// TwinCAT 3 PLC project IBF_Device
// Title: IBF_Device
// Company: Industrial Brains B.V.
// ProjectVersion: 0.0.0.0
// ProgramVersion: 3.1.4022.4
// CompilerDefines: InclSerialCom := 'true'
// libraries:
//   IBF_Utilities, * (Industrial Brains B.V.)
//   Tc2_Math, * (Beckhoff Automation GmbH)
//   Tc2_MC2, * (Beckhoff Automation GmbH)
//   Tc2_MC2_Drive, * (Beckhoff Automation GmbH)
//   Tc2_Standard, * (Beckhoff Automation GmbH)
// project tree:
//   Actuators/Cylinder/DataTypes/ E_CylinderCmd.TcTLEO, E_ValveResetState.TcTLEO (not stored)
//   Actuators/Cylinder/DataTypes/ManualControls/ UDT_ManualValveControl.TcDUT
//   Actuators/Cylinder/Functions/ Fb_DevCylWithFbk.TcPOU (not stored), FB_DevValve.TcPOU (not stored)
//   Axis/DataTypes/ E_AxisCmd.TcTLEO, UDT_AxisData.TcDUT, UDT_AxVal.TcDUT (not stored), UDT_ManualAxisCtrl.TcDUT (not stored)
//   Axis/FunctionBlocks/Analog/ FB_DevAnalogAxis.TcPOU (not stored), ST_ManualAnalogAxisCtrl.TcDUT (not stored)
//   Axis/FunctionBlocks/ServoHybrid/ FB_DevBasicACAxis.TcPOU (not stored), FB_DevHybridAc.TcPOU
//   Axis/FunctionBlocks/Servo/ Fb_DevAxis.TcPOU (not stored)
//   Axis/FunctionBlocks/TwoVelocityControl/DataTypes/ st_ManualDigitalMotorControl.TcDUT (not stored)
//   Axis/FunctionBlocks/TwoVelocityControl/ FB_DevTwoVelocityAxis.TcPOU (not stored)
//   Axis/Interface/ iTwoDirectionalMotor.TcIO (not stored), iTwoDirectionalMotorWithFast.TcIO
//   BaseFunctions/ FB_DevBase.TcPOU (not stored), UDT_DevManualCtrl.TcDUT (not stored)
//   Buttons/Functions/ FB_DevHMIButton.TcPOU, FB_DevPushbuttonLight.TcPOU, FB_DevPushButton.TcPOU
//   CounterCards/FunctionBlocks/KL1512/ FB_DevKL1512.TcPOU (not stored)
//   CounterCards/FunctionBlocks/KL5151/ FB_DevKL5151.TcPOU (not stored)
//   CounterCards/Interfaces/ iCounter.TcIO
//   CounterCards/ st_ManualCounterControl.TcDUT (not stored)
//   DevTypes/ E_Devices.TcTLEO (not stored)
//   Encoders/FunctionBlocks/ FB_EncoderBase.TcPOU (not stored), FB_EncoderInput.TcPOU (not stored)
//   GroupHandlers/ GVL_DevManual.TcGVL (not stored)
//   GroupHandlers/ManualControlHandler/ FB_ManualController.TcPOU (not stored), UDT_DeviceID.TcDUT (not stored)
//   HardwareDiagnostics/ FB_ELModuleDiag.TcPOU (not stored)
//   Heaters/ FB_DevDoublePWM.TcPOU (not stored), FB_DevPWMGenerator.TcPOU (not stored)
//   Lights/Functions/ Fb_DevLight.TcPOU
//   Outputs/AnalogOutputs/ FB_DevAnalogOutput.TcPOU, FB_DevAnalogOutputScaled.TcPOU (not stored)
//   Outputs/DigitalOutputs/ FB_DevDigitalOutput.TcPOU (not stored)
//   Sensors/AnalogInput/FunctionBlocks/ FB_DevAnalogInput.TcPOU (not stored), FB_DevAnalogInputScaled.TcPOU (not stored), FB_DevHDAnalogInAutoCalibrate.TcPOU (not stored), FB_DevAnalogInAutoCalibrate.TcPOU (not stored), FB_DevHDAnalogInputScaled.TcPOU, FB_DevHDAnalogInput.TcPOU (not stored)
//   Sensors/DigitalSensor/FunctionBlocks/ Fb_DevDigitalInput.TcPOU, Fb_DevDigitalInputFunctions.TcPOU (not stored)
//   Sensors/FootPedals/DataTypes/ E_FootpedalPos.TcTLEO (not stored)
//   Sensors/FootPedals/FunctionBlocks/ FB_EfkaEB301A_FootPedal.TcPOU (not stored)
//   Sensors/ModuleSpecific/EL3556_Loadcell/ Fb_DevEL3356_LoadCell.TcPOU
//   Version/ Global_Version.TcGVL

// ---- Actuators/Cylinder/DataTypes/E_CylinderCmd.TcTLEO
(* cylinder commands *)
TYPE E_CylinderCmd :
(
	Cyl_Idle 		:= 0,// Jog Cylinder command Referance 0 Idle (wait for command)
	Cyl_Init 		:= 1,// Jog Cylinder command Referance 1 initialize Cylinder
	Cyl_Enable 		:= 2,// Jog Cylinder command Referance 2 enable
	Cyl_Disable 	:= 3,// Jog Cylinder command Referance 3 disable
	Cyl_Reset 		:= 4,// Jog Cylinder command Referance 4 reset
	Cyl_Hold 		:= 5,// Jog Cylinder command Referance 5 hold
	Cyl_Teach 		:= 6,// Jog Cylinder command Referance 6 teach timeout settings
	Cyl_Calculate 	:= 7,// Jog Cylinder command Referance 7 calculate timeout settings from parameters
	Cyl_Expand 		:= 8,// Jog Cylinder command Referance 8 expand
	Cyl_Retract 	:= 9 // Jog Cylinder command Referance 9 retract
);
END_TYPE

// ---- Actuators/Cylinder/DataTypes/ManualControls/UDT_ManualValveControl.TcDUT
TYPE UDT_ManualValveControl extends UDT_DevManualCtrl:
STRUCT
	// Device commands
	bCmdOpen	: BOOL	; // open valve 
	bCmdClose	: BOOL	; // Close valve
	bCmdTeach	: BOOL	; // Teach valve
END_STRUCT
END_TYPE

// ---- Axis/DataTypes/E_AxisCmd.TcTLEO
(* axis command structure *)
TYPE E_AxisCmd :
(
	Ax_Idle 		:= 0,// Axis command Referance 0 Axis Idle
	Ax_Init 		:= 1,// Axis command Referance 1 Initialize axis
	Ax_Enable 		:= 2,// Axis command Referance 2 Enable
	Ax_Disable 		:= 3,// Axis command Referance 3 Disable
	Ax_Reset 		:= 4,// Axis command Referance 4 Reset
	Ax_Hold 		:= 5,// Axis command Referance 5 Hold
	Ax_Home 		:= 6,// Axis command Referance 6 Home
	Ax_JogFwd 		:= 7,// Axis command Referance 7 Jog Forward
	Ax_JogRev 		:= 8,// Axis command Referance 8 Jog Reverse
	Ax_MoveRelative := 9,// Axis command Referance 9 Move axis relative
	Ax_MoveAbs 		:= 10,// Axis command Referance 11 Move absolute reverse
	Ax_MoveModulo 	:= 11,// Axis command Referance 11 Move Module
	Ax_MoveVeloFwd 	:= 12,// Axis command Referance 12 Move velocity forward
	Ax_MoveVeloRev 	:= 13,// Axis command Referance 13 Move velocity reverse
	Ax_HardStop 	:= 14,// Axis command Referance 14 hard stop or emergency stop
	Ax_SoftStop 	:= 15,// Axis command Referance 15 soft stop after motion command
	Ax_GearSlave 	:= 16,// Axis command Referance 16 gear axis as slave
	Ax_GearSlaveDyn	:= 17,// Axis command Referance 17 gear axis as slave dynamic
	Ax_GearOutSlave := 18,// Axis command Referance 18 gear out from Master axis 
	Ax_Maintenance	:= 50 // Axis Command referance 50 maintenance mode, axis enabled with no command active
);
END_TYPE

// ---- Axis/DataTypes/UDT_AxisData.TcDUT
TYPE UDT_AxisData:
STRUCT
	// ===== Axis name =====
		AxisName	: STRING 	; // Name of the axis (used for fault handling and identification)
		AxisNumber	: INT		; // Axis number 

	// ===== Fault data =====
		Message			: UDT_Fault 	; // Message data from Cylinder
		MessageActive	: BOOL			; // Message is active
		ErrorActive 	: BOOL 			;	// Axis in error state

	// ===== Axis Commands =====
		// ***** Enable command	*****
			CmdEnable		: BOOL 		; // Command enable axis
		// ***** Active commands *****
			AxisCmd			: E_AxisCmd ; // Axis command
			AxisSafeCmd		: E_AxisCmd	; // Axis safe command
			AxisAct			: E_AxisCmd ; // Axis Active status
		// ***** Command Modes *****
			CmdHomingMode 	: MC_HomingMode ; // Homing Mode ( MC_DefaultHoming, MC_Direct, MC_ForceCallibration, MC_ResetCallibration)
			CmdJogMode		: E_JogMode 	;
			CmdBuffermode	: MC_BufferMode	; // Buffermode used for command transition 	 
	// ===== Axis Safe commands =====
		SafeCmdLimitVelo: BOOL 	; // safe command limit velocity
		SafeCmdVelocity	: LREAL ; // Safe command velocity
		SafeCmdStop		: BOOL 	; // Stop command from safety or collision detection		
		SafeVeloLimit	: LREAL ; // safe velocity limit (link to FPAR)
	// ===== Status indication active =====
		ActHoming	: BOOL ; // Axis is homing
		ActBusy		: BOOL ; // Axis is Busy 
		ActMoving	: BOOL ; // Axis is moving
		ActAtVelo	: BOOL ; // Axis is at command velocity (only when written in Move velocity mode)

	// ===== Status indication done  =====
		FcoInit		: BOOL ; // Axis is initialised
		FcoIdle		: BOOL ; // Axis is idle enable required
		FcoEnabled	: BOOL ; // Axis is enabled
		FcoHomed	: BOOL ; // Axis is homed
		FcoGeared	: BOOL ; // Axis is geared to master axis
		FcoHeld		: BOOL ; // Axis is holding
		FcoStopped	: BOOL ; // Axis is stopped
		FcoReset	: BOOL ; // Axis reset done
		FcoReady 	: BOOL ; // Axis is ready for command
		FcoAtCmdPos	: BOOL ; // Axis is at command position (tol 0.2 deg)
		FcoCmdActive: BOOL ; // Axis new command values are active
		
	// ===== Move values =====
		Pos			: UDT_Axval	; // possition values (0 = infinite)
		Velocity 	: UDT_AxVal	; // Velocity values
		Accel		: UDT_Axval ; // Aceleration values
		Decel		: UDT_Axval ; // Deceleration values
		Torque		: UDT_Axval ; // Torque values
		EncTurnoverVal	: DINT 	; // Encoder turnover value
		TimeDisableDelay : TIME ; // Time off delay after axis move command (remove enable)
		
	// ===== Config Bits =====
		IcfCommandSpeedRpm	: BOOL ; // input speeds in Rpm
		IcfEnableForward 	: BOOL ; // Enable forward motion
 		IcfEnablereverse	: BOOL ; // Enable reverse motion
		IcfContinuous		: BOOL ; // continuous motion possible (no endpoint)
		IcfAlwaysEnable		: BOOL ; // 1 = Axis always enabled, 0 = Axis disabled at Idle 
		
	// ===== Master Axis =====
		MasterAxisRef	: REFERENCE TO AXIS_REF ; // Master axis reference (if applicable)
		GearMasterRev	: UINT	:= 1	; // Master Axis Gearing revolutions (Denominator)
		GearSlaveRev	: LREAL	:= 1	; // Slave Axis gearing revolutions (numerator)	
		ReverseSlave	: BOOL 	; // Reverse slave axis relative to master
		 
END_STRUCT
END_TYPE

// ---- Version/Global_Version.TcGVL
{attribute 'TcGenerated'}
{attribute 'no-analysis'}
{attribute 'linkalways'}
// This function has been automatically generated from the project information.
VAR_GLOBAL CONSTANT
	{attribute 'const_non_replaced'}
	stLibVersion_IBF_Device : ST_LibVersion := (iMajor := 0, iMinor := 0, iBuild := 0, iRevision := 0, nFlags := 0, sVersion := '0.0.0.0');
END_VAR

// ---- Axis/Interface/iTwoDirectionalMotorWithFast.TcIO
INTERFACE iTwoDirectionalMotorWithFast EXTENDS iTwoDirectionalMotor // Two directional motor with run fast commands

METHOD CmdRunCCWFast : BOOL
VAR_INPUT
END_VAR
END_METHOD

METHOD CmdRunCWFast : BOOL
VAR_INPUT
END_VAR
END_METHOD

END_INTERFACE

// ---- CounterCards/Interfaces/iCounter.TcIO
INTERFACE iCounter

METHOD PUBLIC CmdResetValue : BOOL
END_METHOD

METHOD PUBLIC CmdSetValue : BOOL
VAR_INPUT
	Value : UDINT ;
END_VAR
END_METHOD

PROPERTY PUBLIC CountValue : UDINT
GET
END_GET
END_PROPERTY

END_INTERFACE

// ---- Axis/FunctionBlocks/ServoHybrid/FB_DevHybridAc.TcPOU
{attribute 'reflection'}
FUNCTION_BLOCK PUBLIC FB_DevHybridAc EXTENDS Fb_DevAxis
VAR_INPUT
END_VAR
VAR_OUTPUT
END_VAR
VAR
	// Parameters 
		stMParMaxAcc : Udt_Parameter := (fMaximum := 999999, fMinimum := 0, fValue := 0)	; // Parameter for maximum acceleration
		stMParMaxDec : Udt_Parameter := (fMaximum := 999999, fMinimum := 0, fValue := 0)	; // Parameter for maximum Deceleration
		stMparMaxVelo: Udt_Parameter := (fMaximum := 999999, fMinimum := 0, fValue := 0)	; // Parameter for maximum velocity
END_VAR

SUPER^(refFbFault := refFbFault);

METHOD INTERNAL ExecHalt : BOOL
VAR_INPUT
END_VAR
// The hybrid axis is equiped with it's own safety stop system therefore mc halt is no longer needed with an Estop
IF bSafetyOk THEN 
	// ==== Execute halt function ===== 
	fbMcHalt (	Axis 		:= AxisRef,
				Execute 	:= bExec_Halt );
END_IF
// ===== reset command =====
	bExec_Halt := FALSE ;
	
// Halt fault handling 
	IF fbMcHalt.Error THEN 
		bError					:= TRUE							;
		stFault.Active 			:= TRUE 						;
		stFault.MessageNumber	:= E_MessageNumbers.FF_AxisFault;
		stFault.Discription		:= CONCAT('Halt Fault ', UDINT_TO_STRING(fbMcHalt.ErrorID));				;
		stFault.FaultType		:= E_FaultTypes.FF				;
	END_IF
END_METHOD

METHOD INTERNAL ExecReadStatus : BOOL
VAR_INPUT
END_VAR
// Read axis status from drive
AxisRef.ReadStatus();						
// convert velocity to RPM for output if aplicable
IF bIcfCmdVelocityRpm THEN 
	fVelocity := AxisRef.NcToPlc.ActVelo / 6 ;
ELSE 
	fVelocity := AxisRef.NcToPlc.ActVelo ;
END_IF

// write position output
fActPosition := AxisRef.NcToPlc.ActPos ;
						
// set status bits 
bIdle := NOT AxisRef.Status.HasJob ;
END_METHOD

METHOD INTERNAL ExecReset : BOOL
VAR_INPUT
END_VAR
IF  AxisRef.Status.Moving AND bExec_Reset THEN // If the axis is still moving execute safe stop first
	CmdSafeStop();
	RETURN;
END_IF

	fbMcReset	( 	Execute	:= bexec_reset,
					Axis	:= AxisRef ); 
					
// ===== reset command =====
	bExec_Reset := FALSE ;
	
// ===== reset internal fault bits and stop bits =====
	bError 			:= FALSE ; 
	
// ===== reset safe commands ======
	bCmdSafeStop	:= FALSE ; 
	bCmdSafeSpeed 	:= FALSE ;
	
// Reset fault handling 
	IF fbMcReset.Error THEN 
		bError					:= TRUE							;
		stFault.Active 			:= TRUE 						;
		stFault.MessageNumber	:= E_MessageNumbers.FF_AxisFault;
		stFault.Discription		:= CONCAT('Reset Fault ', UDINT_TO_STRING(fbMcReset.ErrorID))			;
		stFault.FaultType		:= E_FaultTypes.FF				;
	END_IF
END_METHOD

METHOD PUBLIC Init : BOOL
VAR_INPUT
	// Message location data
	nId			: UDINT ; // Identification number of object
	nParentId	: UDINT ; // Id of higher level If aplicable (0 = no parent)
	// Config Bits
	bIcfCmdVelocityRpm	: BOOL := FALSE ; // input speeds in Rpm
	bIcfEnableForward 	: BOOL := TRUE 	; // Enable forward motion
	bIcfEnablereverse	: BOOL := TRUE 	; // Enable reverse motion
	bIcfAlwaysEnable	: BOOL := FALSE ; // 1 = Axis always enabled, 0 = Axis disabled at Idle 
	bIcfSimulationMode	: BOOL := FALSE ; // Simulation mode is active [default set to False] Used for testing without hardware present 
	bIcfModuloAxis		: BOOL := FALSE ; // Show axis position as modulo
	bIcfSTOPresent		: BOOL := FALSE ; // Axis safe torque off is present	
	bIcfNCHomeSensor	: BOOL := FALSE ; // Homing sensor is inverted (NC)	

	// Config Values 
	mcHomingMode 		: MC_HomingMode := MC_HomingMode.MC_DefaultHoming; 
	fHomePosition		: LREAL := 0 	; // set position at homing
	fSafeOverride		: LREAL := 10	; // Safe velocity override [%]
	nEncTurnoverVal 	: LREAL := 360	; // encoder turnover value 
	tEnableDelay		: time 	:= T#0MS; // Time between axis enable command and motion command execution (0 := no delay active)	
	tDisabledelay		: TIME 	:= T#100MS; // Axis idle time before axis is disabled 
END_VAR
VAR 
	bActVeloReadValid 	: BOOL ; // velocity parameter read is valid 
	bActAccReadValid 	: BOOL ; // Acceleration parameter read is valid 
	bActDecReadValid 	: BOOL ; // Deceleration parameter read is valid 
	bActParamValid 		: BOOL ; // Parameter read is valid 
END_VAR
// Calculate device number
	ExecIdentifyDevice(nId,nParentId, E_ComponentTypes.Axis);

// ===== Message data set =====
	stFault.ComponentType		:= E_ComponentTypes.Axis ;
	
// ===== Write parameters =====
	stMParMaxAcc.nNumber		:= nLocationId + 1;
	stMParMaxAcc.sDiscription 	:= CONCAT(STR1 := sName, STR2:= ' hardware maximum accaleration (0 = HWMaximum)'); 
	stMParMaxAcc.sName			:= CONCAT(STR1 := sName, STR2:= 'Hard max aceleration');
	stMParMaxAcc.sType			:= 'MPar';
	stMParMaxAcc.sUnit			:= 'Units/Sec^2';
	
	stMParMaxDec.nNumber		:= nLocationId + 2;
	stMParMaxDec.sDiscription 	:= CONCAT(STR1 := sName, STR2:= ' hardware maximum deceleration(0 = HWMaximum)'); 
	stMParMaxDec.sName			:= CONCAT(STR1 := sName, STR2:= 'Hard max deceleration');
	stMParMaxDec.sType			:= 'MPar';
	stMParMaxDec.sUnit			:= 'Units/Sec^2';
	
	stMparMaxVelo.nNumber		:= nLocationId + 3;
	stMparMaxVelo.sDiscription 	:= CONCAT(STR1 := sName, STR2:= ' hardware maximum velocity'); 
	stMparMaxVelo.sName			:= CONCAT(STR1 := sName, STR2:= 'Hard max velocity');
	stMparMaxVelo.sType			:= 'MPar';
	stMparMaxVelo.sUnit			:= 'Units/Sec';

	refFbParHandler.CmdAddParameter(refParameter := stMParMaxAcc);
	refFbParHandler.CmdAddParameter(refParameter := stMParMaxDec);
	refFbParHandler.CmdAddParameter(refParameter := stMparMaxVelo);

// ===== set axis configuration =====	
	fMaxAcc	:= stMParMaxAcc.fValue;
	fMaxDec	:= stMParMaxDec.fValue;	
	fMaxVelo:= stMparMaxVelo.fValue;

	fCmdAcc 		:= fMaxAcc;
	fCmdDecc		:= fMaxDec;
// ===== Configure Axis =====
	// ***** Config Bits *****
		THIS^.bIcfCmdVelocityRpm	:= bIcfCmdVelocityRpm	; // Enable speed inputs in Rpm
		THIS^.bIcfEnableForward 	:= bIcfEnableForward 	; // Enable forward motion
		THIS^.bIcfEnablereverse		:= bIcfEnablereverse	; // Enable reverse motion
		THIS^.bIcfAlwaysEnable		:= bIcfAlwaysEnable		; // Always enable motor and brake if safety is ok
		THIS^.bIcfSimulationMode	:= bIcfSimulationMode 	; // Simulation mode is active [default set to False] 

	// ***** config homing Mode ***** 
 		THIS^.mcHomingMode 			:= mcHomingMode ; // set homing mode
 		THIS^.fHomePosition			:= fHomePosition;
	// ***** Velocity settings *****
		THIS^.fSafeOverride			:= fSafeOverride	; 	
	// ***** Time delay enable off *****
		THIS^.tEnableDelay		:= tEnableDelay	;
		THIS^.tDisableDelay 	:= tDisabledelay ;		

// ===== Set device type for manual control =====
	eDevType := E_Devices.Axis ;
		
// ===== reset axis state indicators ======
	bErrorActive 	:= FALSE;

// ====== Set init to done =======
	bInitOk	:= TRUE ;
END_METHOD

END_FUNCTION_BLOCK

// ---- Buttons/Functions/FB_DevHMIButton.TcPOU
{attribute 'reflection'}
FUNCTION_BLOCK PUBLIC FB_DevHMIButton EXTENDS FB_DevBase // Button function for HMI 
VAR_INPUT
	Istatus			: BOOL	:= FALSE;// Digital sensor, Direct input status
	tDelay			: TIME 	:= T#5S	;// Time before delayed signal becomes active 
END_VAR
VAR_OUTPUT
	bFcoInputActive		: BOOL 			;// Digital sensor, Button active state
	bFcoDelay			: BOOL			;// Button, Delayed input status (3 seconds) 
	bFeStatus			: BOOL			;// Button, Falling edge of input signal	
	bReStatus			: BOOL			;// Button, Rising edge of input signal
	TetInputActive		: TIME			;// Button, Time elapsed while button is active
	bInvisible			: BOOL 			;// Button, Button is made invisible
	bDeactivate			: BOOL 			;// Button, Deactivate button 
END_VAR
VAR
	FB_delIStatus	: TON; // Timer function for delayed input status 
	FB_feIStatus	: F_TRIG; // generate falling edge pulse edge from Istatus
	FB_reIStatus	: R_TRIG; // generate falling edge pulse edge from Istatus
END_VAR

// Call base function
SUPER^(refFbFault := refFbFault);

// ***** Direct input when enabled *****
IF bEnable THEN 
	bFcoInputActive := Istatus ;
ELSE 
	bFcoInputActive := FALSE ;
END_IF

// ===== check if function is enabled =====
	IF NOT bEnable THEN 
		bInvisible 	:= TRUE ;
		bDeactivate	:= TRUE ;
		bFcoDelay	:= FALSE;
		RETURN;
	ELSE  
		bInvisible 	:= FALSE ;
		bDeactivate	:= FALSE ;
	END_IF

// ====== process functions if enabled ======
	// ***** Set Delayed inputs and time elapsed ****
		FB_delIStatus(	IN:= bFcoInputActive,
						PT:= tDelay , 
						Q=> bFcoDelay , 
						ET=> TetInputActive 
					  ); // Generate delayed input status from push button input status
	// ***** Edge triggers *****
		FB_feIStatus(CLK:= Istatus , Q=> bFeStatus ); // generate falling edge pulse on pushbutton input
		FB_reIStatus (Clk := Istatus , Q => bReStatus); // Generate rising edge from push button input signal

END_FUNCTION_BLOCK

// ---- Buttons/Functions/FB_DevPushbuttonLight.TcPOU
{attribute 'reflection'}
FUNCTION_BLOCK PUBLIC FB_DevPushbuttonLight EXTENDS Fb_DevDigitalInputFunctions
VAR_OUTPUT
END_VAR
VAR
	fbLight : Fb_DevLight ; // light control 
END_VAR

// Set device type
IF eDevType = E_Devices.Undefined THEN 
	eDevType := E_Devices.PushButtonLight ;
END_IF

SUPER^(refFbFault := refFbFault);

// Light commands
	
fbLight(bEnable := bEnable, refFbFault := refFbFault);

METHOD PUBLIC CmdBlinkFast : BOOL
VAR_INPUT
END_VAR
CmdBlinkFast := fbLight.CmdBlinkFast();
END_METHOD

METHOD PUBLIC CmdBlinkSlow : BOOL
VAR_INPUT
END_VAR
CmdBlinkSlow	:= fbLight.CmdBlinkSlow();
END_METHOD

METHOD PUBLIC CmdOn : BOOL
VAR_INPUT
END_VAR
CmdOn := fbLight.CmdOn() ;
END_METHOD

END_FUNCTION_BLOCK

// ---- Lights/Functions/Fb_DevLight.TcPOU
{attribute 'reflection'}
FUNCTION_BLOCK PUBLIC Fb_DevLight EXTENDS FB_DevBase ;
VAR_OUTPUT
	bSoftLightOut	: BOOL ; // Software light output	
END_VAR
VAR
	bCmdBlinkSlow	: BOOL := FALSE ; // Command light blink slow
	bCmdBlinkFast 	: BOOL := FALSE ; // Command light blink fast
	bCmdOn			: BOOL := FALSE ; // Command turn light on	 
	qLight AT %Q* 	: BOOL := FALSE ; // light output
END_VAR

// set device type
IF eDevType = E_Devices.Undefined THEN 
	eDevType := E_Devices.DigitalOut ;
END_IF

// ===== check if light is enabled ======
	IF NOT bEnable AND NOT bCmdManual THEN 
		qLight := FALSE ;
		RETURN; 
	END_IF
	
// ===== set light output ======
	ExecSetOutput();

METHOD PUBLIC CmdBlinkFast : BOOL
VAR_INPUT
END_VAR
bCmdBlinkFast S= TRUE ;

CmdBlinkFast := bCmdBlinkFast ;
END_METHOD

METHOD PUBLIC CmdBlinkSlow : BOOL
VAR_INPUT
END_VAR
bCmdBlinkSlow S= TRUE ;

CmdBlinkSlow	:= bCmdBlinkSlow ;
END_METHOD

METHOD PUBLIC CmdOn : BOOL
VAR_INPUT
END_VAR
bCmdOn S= TRUE ;

CmdOn := qLight ;
END_METHOD

METHOD PRIVATE ExecSetOutput : BOOL
VAR_INPUT
END_VAR
// ===== set light output state =====
IF bCmdOn THEN 
	qLight S= TRUE ;
ELSIF bCmdBlinkFast THEN 
	qLight := Sys_Variables.BlinkFast 	;
ELSIF bCmdBlinkSlow THEN 
	qLight := Sys_Variables.BlinkSlow	;
ELSE
	qLight := FALSE ;
END_IF

// set soft output
bSoftLightOut	:= qLight;

// reset all commands 
bCmdOn			:= FALSE ;
bCmdBlinkFast 	:= FALSE ;
bCmdBlinkSlow 	:= FALSE ;
END_METHOD

METHOD PUBLIC Init : BOOL
VAR_INPUT
	// Location data for messages  
	nId			: UDINT ; // Identification number of object
	nParentId	: UDINT ; // Id of higher level If aplicable (0 = no parent)
END_VAR
// ====== Set init to true =====
	bInitOk	:= TRUE ; 

// ====== Calculate device id =====
	bInitOk :=	ExecIdentifyDevice(nId,nParentId, E_ComponentTypes.DiOutput) AND bInitOk;

// ===== Set feedback =====
	Init := bInitOk;
END_METHOD

END_FUNCTION_BLOCK

// ---- Buttons/Functions/FB_DevPushButton.TcPOU
{attribute 'reflection'}
FUNCTION_BLOCK PUBLIC FB_DevPushButton EXTENDS Fb_DevDigitalInputFunctions
VAR_INPUT
END_VAR
VAR_OUTPUT
END_VAR
VAR
END_VAR

// set device type
IF eDevType = E_Devices.Undefined THEN 
	eDevType := E_Devices.DigitalSensor ;
END_IF

SUPER^(refFbFault := refFbFault);

END_FUNCTION_BLOCK

// ---- Outputs/AnalogOutputs/FB_DevAnalogOutput.TcPOU
{attribute 'reflection'}
FUNCTION_BLOCK PUBLIC FB_DevAnalogOutput EXTENDS FB_DevBase 
VAR_INPUT
	fCmdValue		: LREAL := 0 ;
END_VAR
VAR_OUTPUT
	fOutputValue	: LREAL := 0 ;
END_VAR
VAR
	nLimitMin		: INT := -32767 ;
	nLimitMax 		: INT := 32767 ;
	qnHwOut	AT%Q*	: INT := 0 ;
END_VAR

// set device type
IF eDevType = E_Devices.Undefined THEN 
	eDevType := E_Devices.AnalogOut ;
END_IF

// Call base function
SUPER^(refFbFault := refFbFault);


// Call private functions
ExecSetOutput();
ExecSetFeedback();

METHOD INTERNAL ExecSetFeedback : BOOL
VAR_INPUT
END_VAR
// Set feedback 
fOutputValue := INT_TO_LREAL(qnHwOut) ;
END_METHOD

METHOD INTERNAL ExecSetOutput : BOOL
VAR_INPUT
END_VAR
// Set Output to physical device
IF bSafetyOk AND (bEnable OR bCmdManual) THEN 
	qnHwOut := LREAL_TO_INT(fCmdValue) ; 
	qnHwOut := LIMIT(nLimitMin, qnHwOut, nLimitMax) ; 
ELSE 
	qnHwOut 	:= 0;
	fCmdValue 	:= 0 ; 
END_IF
END_METHOD

METHOD PUBLIC Init : BOOL
VAR_INPUT
	// Location data for messages  
	nId				: UDINT; // Identification number of object
	nParentId		: UDINT; // Id of higher level If aplicable (0 = no parent)
	benableNegative	: BOOL ; // Enable negative values
END_VAR
// ====== Set init to true =====
	bInitOk	:= TRUE ; 

// ====== Calculate device id =====
	bInitOk :=	ExecIdentifyDevice(nId,nParentId, E_ComponentTypes.AnOutput) AND bInitOk;
	
// ====== set minimum value ========
	IF benableNegative THEN 
		nLimitMin := -32767;
	ELSE
		nLimitMin := 0 ;
	END_IF
	
// ====== Set feedback ======
	Init 	:= TRUE ;
END_METHOD

END_FUNCTION_BLOCK

// ---- Sensors/AnalogInput/FunctionBlocks/FB_DevHDAnalogInputScaled.TcPOU
{attribute 'reflection'}
FUNCTION_BLOCK PUBLIC FB_DevHDAnalogInputScaled EXTENDS FB_DevHDAnalogInput
VAR_INPUT
END_VAR
VAR_OUTPUT
END_VAR
VAR
	fGainFactor 	: LREAL	:= 1	;
	nOfset			: DINT	:= 0	;
END_VAR

SUPER^(refFbFault := refFbFault);

METHOD ExecSetFeedback : BOOL
VAR
	nCalibValue	: DINT ; 
END_VAR
// Offset 
IF bCmdSimulate THEN 
	nCalibValue := fSimValue + nOfset ;
ELSE
	nCalibValue := inHwInput + nOfset ;
END_IF

fValue := DINT_TO_LREAL(nCalibValue) / fGainFactor;

ExecSetFeedback := TRUE;
END_METHOD

METHOD PUBLIC SetScaling : BOOL 
VAR_INPUT
	fMaxValue	: LREAL ; 	// Maximum input value after scaling, e.g. 100%, 0 = no scaling (gain = hardware limit / fMaxValue)  
	fOfset		: LREAL ;	// offset value (fvalue = (gain * hwvalue) + fOfset)
END_VAR
// calculate gain 
IF fMaxValue =0 THEN 
	fGainFactor := 1 ;
ELSE 
	fGainFactor := nLimitMax / fMaxValue ;
END_IF

nOfset := LREAL_TO_DINT(fOfset * fGainFactor) ;

SetScaling := TRUE;
END_METHOD

END_FUNCTION_BLOCK

// ---- Sensors/DigitalSensor/FunctionBlocks/Fb_DevDigitalInput.TcPOU
{attribute 'reflection'}
FUNCTION_BLOCK PUBLIC Fb_DevDigitalInput EXTENDS FB_DevBase 
VAR_INPUT
	tDelay				: TIME 	:= T#1S	;// Time before delayed signal becomes active 
	bCmdSimulate		: BOOL 	:= FALSE ;// Simulate sensor Input 
	bSimState			: BOOL 	:= FALSE ;// Simulated sensor state
	bIcfNormalyClosed	: BOOL  := FALSE ;// Hardware input is a normally closed contact
	ibSoftInput			: BOOL 			;// Software input (bFcoInputActive := 
END_VAR
VAR_OUTPUT
	bFcoInputActive		: BOOL 			;// Digital sensor, Button active state
END_VAR
VAR
	Istatus		AT 	%I* : BOOL			;// Digital sensor, Direct input status
END_VAR

// Set device type
IF eDevType = E_Devices.Undefined THEN 
	eDevType := E_Devices.DigitalSensor ;
END_IF

// Call base function
SUPER^(refFbFault := refFbFault);

// ***** Direct input when enabled *****
IF bEnable OR bCmdManual THEN 
	IF bCmdSimulate  THEN 
		bFcoInputActive := bSimState ;
		bCmdSimulate	:= FALSE ;  
	ELSIF bIcfNormalyClosed THEN
		bFcoInputActive := NOT Istatus OR ibSoftInput;
	ELSE
		bFcoInputActive := Istatus OR ibSoftInput ;
	END_IF
ELSE 
	bFcoInputActive := FALSE ;
END_IF

METHOD PUBLIC Init : BOOL
VAR_INPUT
	// Location data for messages  
	nId			: UDINT ; // Identification number of object
	nParentId	: UDINT ; // Id of higher level If aplicable (0 = no parent)
END_VAR
// ====== Set init to true =====
	bInitOk	:= TRUE ; 

// ====== Calculate device id =====
	bInitOk :=	ExecIdentifyDevice(nId,nParentId, E_ComponentTypes.DiInput) AND bInitOk;

	Init	:= true ;
END_METHOD

END_FUNCTION_BLOCK

// ---- Sensors/ModuleSpecific/EL3556_Loadcell/Fb_DevEL3356_LoadCell.TcPOU
FUNCTION_BLOCK PUBLIC Fb_DevEL3356_LoadCell EXTENDS FB_DevHDAnalogInAutoCalibrate
VAR_INPUT
	tCalibrationDelay	: TIME := T#2S ; // Time for which the load neads to before calibration is done (default T#2s) 
END_VAR
VAR_OUTPUT
	bMeasurementError	: BOOL 		; // Measurement or component error is active
	sErroDiscription 	: STRING 	; // 
END_VAR
VAR
	ibOverrange				AT%I*	: BOOL ; // overrange status indication
	ibDataInvalid			AT%I*	: BOOL ; // Data is invalid
	ibError					AT%I*	: BOOL ; // Module is in error state
	ibCalibrationinProgress	AT%I*	: BOOL ; // automatic calibration is in progress
	ibSteadyState			AT%I*	: BOOL ; // Module is in steady state
	ibSyncError				AT%I*	: BOOL ; // Module sync error
	
	tonSteadyState	: TON ; // steady state delay for calibration
END_VAR

ACTION CheckELSignalState:
// Set error device measurement error bit
bMeasurementError := FALSE ;

IF ibOverrange THEN 
	bMeasurementError 	S= TRUE;
 	sErroDiscription	:= 'Load exceeds maximum range ';
ELSIF ibDataInvalid THEN
	bMeasurementError 	S= TRUE;
	sErroDiscription	:= 'Incorrect date from device';
ELSIF ibError THEN
	bMeasurementError 	S= TRUE;
	sErroDiscription	:= 'Module general error';
ELSIF ibCalibrationinProgress THEN
	bMeasurementError 	S= TRUE;
	sErroDiscription	:= 'Calibration session in progress';
ELSIF ibSyncError THEN
	bMeasurementError 	S= TRUE;
	sErroDiscription	:= 'Module ethercat sync error';	
END_IF
END_ACTION

METHOD PUBLIC CmdCalibrateNull : BOOL
VAR_INPUT
END_VAR
tonSteadyState(IN := ibSteadyState, PT := tCalibrationDelay);

// set offset to calibrate to null
IF tonSteadyState.Q THEN 
	nOfset := - inHwInput ;
END_IF
END_METHOD

METHOD PUBLIC CmdCalilbrateValue : BOOL // calibrate gain factor to actual value (warning calibrate to null before calibrating to value)
VAR_INPUT
	fCalibrationValue	: LREAL ; // Active input value to sensor [N]
END_VAR
tonSteadyState(IN := ibSteadyState, PT := tCalibrationDelay);

// set gain from current value
IF tonSteadyState.Q THEN 
	fGainFactor := DINT_TO_LREAL(inHwInput + nOfset) / fCalibrationValue ; 
END_IF
END_METHOD

END_FUNCTION_BLOCK
